TYPE DUT_cfgPosicValvula :
STRUCT
	//Essa struct estrutura os parâmetros de conversão do posicionamento das válvulas
	Aberta	:INT;
	Fechada	:INT;
END_STRUCT
END_TYPE

(* stored: Version 1.1.0.1, ProductVersion 3.1.4024.14
   DUT DUT_cfgPosicValvula: Id {499987a9-a48c-4a42-a6f1-daabb7c85afc} *)
